// TIA Portal V17 export
// export: Created 2023-02-14T02:49:31.9929696Z, ExportSetting WithDefaults, DisplayName Totally Integrated Automation Portal, DisplayVersion V17, DisplayName TIA Portal Openness, DisplayVersion V17, DisplayName TIA Portal Teamcenter Gateway, DisplayVersion V17, DisplayName TIA Portal Version Control Interface, DisplayVersion V17, DisplayName SINAMICS Startdrive Advanced, DisplayVersion V17, DisplayName SINAMICS Startdrive G130, G150, S120, S150, SINAMICS MV, S210, DisplayVersion V17, DisplayName SINAMICS Startdrive G110M, G120, G120C, G120D, G120P, G115D, DisplayVersion V17, DisplayName STEP 7 Professional, DisplayVersion V17, DisplayName STEP 7 Safety, DisplayVersion V17, DisplayName WinCC Professional, DisplayVersion V17
DATA_BLOCK "IO Motor MCC Preparation_DB"   // DB12
VERSION : 0.1
// stored: AutoNumber true, DBAccessibleFromOPCUA true, DBAccessibleFromWebserver true, InstanceOfName IO Motor MCC Preparation, InstanceOfType FB
"IO Motor MCC Preparation"
   // VAR_INPUT
   //    lock : Bool;
   //    Init : Bool;
   //    EM_Stop : Bool;
   //    Testing : Bool;
   //    Reset : Bool;
   // END_VAR
   // VAR
   //    "P-01.01" { S7_SetPoint := 'True'} : "Motor_w_VSD";
   //    "P-02.01" { S7_SetPoint := 'True'} : "Motor_w_VSD";
   //    "P-02.03" { S7_SetPoint := 'True'} : "Motor_w_VSD";
   //    "P-03.01" { S7_SetPoint := 'True'} : "Motor_w_VSD";
   //    "P-03.03" { S7_SetPoint := 'True'} : "Motor_w_VSD";
   //    "P-04.01" { S7_SetPoint := 'True'} : "Motor_w_VSD";
   //    "XA-05.01" { S7_SetPoint := 'True'} : "Motor_w_VSD";
   //    "P-05.01" { S7_SetPoint := 'True'} : "Motor_w_VSD";
   //    "P-05.03_DOL" { S7_SetPoint := 'True'} : "Motor";
   //    "P-06.01" { S7_SetPoint := 'True'} : "Motor_w_VSD";
   //    "P-07.01" { S7_SetPoint := 'True'} : "Motor_w_VSD";
   //    "P-08.01" { S7_SetPoint := 'True'} : "Motor_w_VSD";
   //    "P-08.02" { S7_SetPoint := 'True'} : "Motor_w_VSD";
   //    "XA-09.01" { S7_SetPoint := 'True'} : "Motor_w_VSD";
   //    "P-09.01" { S7_SetPoint := 'True'} : "Motor_w_VSD";
   //    "P-09.03" { S7_SetPoint := 'True'} : "Motor";
   //    "P-10.01" { S7_SetPoint := 'True'} : "Motor_w_VSD";
   //    "P-51.01" { S7_SetPoint := 'True'} : "Motor_w_VSD";
   // END_VAR
BEGIN
END_DATA_BLOCK
